// TIA Portal V20 export
DATA_BLOCK "T5 EXCENTRIC LEV2"   // DB1718
{ S7_Optimized_Access := 'TRUE' }
AUTHOR : SAS
// stored: AutoNumber false, IsRetainMemResEnabled true, MemoryReserve 100, RetainMemoryReserve 100
   VAR RETAIN
      ITF : Struct
         "Production Lock" : Bool;
         "Check OK" : Bool;
         "Check not OK" : Bool;
         "Transfer OK" : Bool;
         "Transfer not OK" : Bool;
         Skip : Bool;   // Coupling not to work (0=to work, 1= not to work)
         Status : Int;
      END_STRUCT;
      MEMORY : Struct
         PP_Man_Mov : Bool;   // Pipe presence for manual movement
         "Cond move Fwd" : Bool;   // Cond move Fwd
         "Unlock LEV.2 ANSWER" : Bool;   // Unlock LEV.2 ANSWER (1=Unlock)
         CheckRequestMemory : Bool;   // Tracking Check request memory
      END_STRUCT;
   END_VAR
   VAR
      SEQ { S7_SetPoint := 'True'} : "SEQ LIV2";
      AUX : Struct
         "TIMER" { S7_SetPoint := 'True'} : Array[1..50] of IEC_TIMER;
         OS : Array[0..50] of Bool;
      END_STRUCT;
   END_VAR
BEGIN
   // SEQ.SEQ.S01 : STARTUP
   // SEQ.SEQ.S28 : FINE
   // SEQ.SEQ.S29 : MANUALE
   // SEQ.SEQ.S30 : FAULT
   // SEQ.SEQ.S32 : EMERGENZA
END_DATA_BLOCK
